KUKA KRL data list: Wood_Test_2.dat

&ACCESS RVEO
&REL 38
&PARAM DISKPATH = KRC:\R1\Program\Milling
DEFDAT  WOOD_TEST_2 PUBLIC

DECL AXIS lAstartPos={A1 -22.4984303,A2 -99.5414124,A3 132.718292,A4 75.8801346,A5 -68.2717209,A6 -55.2195663}
DECL FRAME lfPrePos[5]
lfPrePos[1]={X -32.0000,Y -50.0000,Z 350.000,A 90.0000,B 0.0,C -45.0000}
lfPrePos[2]={X -32.0000,Y -15.0000,Z 70.0000,A 90.0000,B 0.0,C -90.0000}
lfPrePos[3]={X 0.0,Y -32.0000,Z 70.0000,A 0.0,B 0.0,C 90.0000}
lfPrePos[4]={X 0.0,Y -32.0000,Z 50.0000,A 90.0000,B 0.0,C 0.0}
lfPrePos[5]={X 0.0,Y -50.0000,Z 350.000,A 90.0000,B 0.0,C 0.0}

DECL FRAME lfWorkPos[12]
lfWorkPos[1]={X 0.0,Y 180.000,Z 0.0,A 0.0,B 0.0,C 0.0}
lfWorkPos[2]={X 0.0,Y -40.0,Z 0.0,A 0.0,B 0.0,C 0.0}
lfWorkPos[3]={X 0.0,Y 0.0,Z 0.0,A 0.0,B 0.0,C 90.0000}
lfWorkPos[4]={X 0.0,Y 200.000,Z 0.0,A 0.0,B 0.0,C 90.0000}

lfWorkPos[5]={X 12.5000,Y 340.000,Z 0.0,A 0.0,B 0.0,C 0.0}
lfWorkPos[6]={X 12.5000,Y 12.5000,Z 0.0,A 0.0,B 0.0,C 0.0}
lfWorkPos[7]={X 200.000,Y 12.5000,Z 0.0,A 0.0,B 0.0,C 0.0}

lfWorkPos[8]={X 200.000,Y 1.00000,Z 0.0,A 0.0,B 0.0,C 45.0000}
lfWorkPos[9]={X 0.0,Y 1.00000,Z 0.0,A 0.0,B 0.0,C 45.0000}
lfWorkPos[10]={X 1.00000,Y 0.0,Z 0.0,A 0.0,B -45.0000,C 0.0}
lfWorkPos[11]={X 1.00000,Y 200.000,Z 0.0,A 0.0,B -45.0000,C 0.0}
ENDDAT
